{attribute 'qualified_only'}
VAR_GLOBAL
END_VAR

(* stored: Version 1.1.0.1, ProductVersion 3.1.4024.13
   GVL Hardware_Mapping: Id {5e079435-37e1-4dac-9ffd-d7430a992c47} *)
